// TwinCAT 3 PLC project NewPort_Stepper
// ProgramVersion: 3.1.4023.0
// libraries:
//   Tc2_Standard, * (Beckhoff Automation GmbH)
//   Tc2_System, * (Beckhoff Automation GmbH)
//   Tc3_Module, * (Beckhoff Automation GmbH)
// project tree:
//   / PlcTask.TcTTO
//   POUs/ MAIN.TcPOU
// real-time tasks:
//   TASK PlcTask: cycle T#10ms, priority 20, ADS port 350
// motion (NC):
//   TASK NC-Task 1 SAF: cycle T#2ms, priority 4, ADS port 501
//   TASK NC-Task 1 SVB: cycle T#10ms, priority 8, ADS port 511
//   AXIS Axis 1 (id 1)
//     Dynamic: AccelerationMaximum=1, DecelerationMaximum=1, Acceleration=1, Deceleration=1, Jerk=1.2
//     Velo: RefSearch=0.1, RefSync=0.1, SlowManual=0.2, FastManual=0.2, Maximum=0.4
//     OtherSettings: AllowMotionCmdToSlave=true, PulseDistancePos=0.1, PulseDistanceNeg=0.1
//     encoder EncType=4
//       EncPara: ScaleFactorNumerator=1.52587e-06, MaxCount=#xffffffff
//         Inc: RefSoftSyncMask=#x0000ffff
//     drive DrvType=24
//       Analog: VeloReferenz=0.4, TorqueSetpointScale=10, ScaleFactorActTorque=0.1
//       TimeComp: TaskDelayCycles=1
//     controller CtrType=1
//       CtrPara: PriorControlFactor=1
//         Observer: BandWidth=20
// I/O:
//   DEVICE Device 2 (EtherCAT), AmsNetId 10.33.178.144.3.1
//     Term 1 (EK1101) [EK1101 EtherCAT Coupler (2A E-Bus, ID switch)]
//       Term 2 (EL7041) [EL7041 1Ch. Stepper motor output stage (50V, 5A)]
//       Term 3 (EL6022) [EL6022 Interface 2Ch. (RS422/485)]
//       Term 4 (EL9011) [EL9011 End Terminal]
// variable links:
//   NC-Task 1 SAF/Axes/Axis 1 <-> Device 2 (EtherCAT)/Term 1 (EK1101)/Term 2 (EL7041)
//     Drive/Inputs/In/nState1 @bit 3 <-> STM Status/Status/Error
//     Drive/Inputs/In/nState1 @bit 5 <-> STM Status/Status/Moving negative
//     Drive/Inputs/In/nState1 @bit 4 <-> STM Status/Status/Moving positive
//     Drive/Inputs/In/nState1 @bit 1 <-> STM Status/Status/Ready
//     Drive/Inputs/In/nState1 <-> STM Status/Status/Ready to enable
//     Drive/Inputs/In/nState1 @bit 6 <-> STM Status/Status/Torque reduced
//     Drive/Inputs/In/nState1 @bit 2 <-> STM Status/Status/Warning
//     Drive/Inputs/In/nState2 @bit 3 <-> STM Status/Status/Digital input 1
//     Drive/Inputs/In/nState2 @bit 4 <-> STM Status/Status/Digital input 2
//     Drive/Inputs/In/nState2 @bit 5 <-> STM Status/Status/Sync error
//     Drive/Inputs/In/nState2 @bit 7 <-> STM Status/Status/TxPDO Toggle
//     Drive/Inputs/In/nState4 @bit 1 <-> WcState/InputToggle
//     Drive/Inputs/In/nState4 <-> WcState/WcState
//     Drive/Outputs/Out/nCtrl1 <-> STM Control/Control/Enable
//     Drive/Outputs/Out/nCtrl1 @bit 2 <-> STM Control/Control/Reduce torque
//     Drive/Outputs/Out/nCtrl1 @bit 1 <-> STM Control/Control/Reset
//     Enc/Inputs/In/nDataIn1 <-> ENC Status/Counter value
//     Enc/Inputs/In/nDataIn2 <-> ENC Status/Latch value
//     Enc/Inputs/In/nState1 @bit 4 <-> ENC Status/Status/Counter overflow
//     Enc/Inputs/In/nState1 @bit 3 <-> ENC Status/Status/Counter underflow
//     Enc/Inputs/In/nState1 @bit 7 <-> ENC Status/Status/Extrapolation stall
//     Enc/Inputs/In/nState1 <-> ENC Status/Status/Latch C valid
//     Enc/Inputs/In/nState1 @bit 1 <-> ENC Status/Status/Latch extern valid
//     Enc/Inputs/In/nState1 @bit 2 <-> ENC Status/Status/Set counter done
//     Enc/Inputs/In/nState2 @bit 4 <-> ENC Status/Status/Status of extern latch
//     Enc/Inputs/In/nState2 <-> ENC Status/Status/Status of input A
//     Enc/Inputs/In/nState2 @bit 1 <-> ENC Status/Status/Status of input B
//     Enc/Inputs/In/nState2 @bit 2 <-> ENC Status/Status/Status of input C
//     Enc/Inputs/In/nState2 @bit 5 <-> ENC Status/Status/Sync error
//     Enc/Inputs/In/nState2 @bit 7 <-> ENC Status/Status/TxPDO Toggle
//     Enc/Inputs/In/nState4 @bit 1 <-> WcState/InputToggle
//     Enc/Inputs/In/nState4 <-> WcState/WcState
//     Enc/Outputs/Out/nCtrl1 <-> ENC Control/Control/Enable latch C
//     Enc/Outputs/Out/nCtrl1 @bit 3 <-> ENC Control/Control/Enable latch extern on negative edge
//     Enc/Outputs/Out/nCtrl1 @bit 1 <-> ENC Control/Control/Enable latch extern on positive edge
//     Enc/Outputs/Out/nCtrl1 @bit 2 <-> ENC Control/Control/Set counter
//     Enc/Outputs/Out/nDataOut1 <-> ENC Control/Set counter value

CONFIGURATION NewPort_Stepper
    RESOURCE PLC ON TwinCAT3
        TASK PlcTask(INTERVAL := T#10ms, PRIORITY := 20);
        PROGRAM MAIN WITH PlcTask : MAIN;
    END_RESOURCE
END_CONFIGURATION

// ---- POUs/MAIN.TcPOU
PROGRAM MAIN
VAR
END_VAR

END_PROGRAM
